FUNCTION "_outOfRangeWithDelay" : Bool
TITLE = {"status":"current","deprecatedBy": null,"dependencies" : ["TON_TIME"]}
{ S7_Optimized_Access := 'TRUE' }
AUTHOR : cyanezf
FAMILY : 'core/control/util'
NAME : _outOfRangeWithDelay
VERSION : 1.1

   VAR_INPUT
      homed : Bool;   // 1=Homed and sync ok (if there are sync axis)
      actualPosition : LReal;   // Actual position
      minPosition : LReal;   // Min reference position
      maxPosition : LReal;   // Max reference position
      tolerance : LReal;   // Tolerance (Add this value to position)
      delay : Time;   // Delay time
   END_VAR

   VAR_IN_OUT
      "timer" {InstructionName := 'TON_TIME'; LibVersion := '1.0'} : TON_TIME;   // Delay timer
   END_VAR

BEGIN
(*--
# Documentation

## Log

| version | date | author | description |
|:-------:|:----:|:------:|:------------|
| v1.1 | 2026-06-17 | cyanezf | refactor: Change REAL to LREAL  |
| v1.0 | 2026-05-12 | cyanezf | First version |

## Description

This function checks if the `actualPosition` is out of range with tolerance and is homed.

--*)

	#timer(IN := #homed AND #actualPosition < #minPosition + #tolerance AND #actualPosition > #maxPosition - #tolerance,
	       PT := #delay);

	// Save RLO
	ENO := #_outOfRangeWithDelay := #timer.Q;

END_FUNCTION

